TYPE (* A cloud representation for the Arrowhead framework 4.0 *)
  (* Standard: 61499-2 *)
  (* Version 1.0, 2018-09-26, Jose Cabral, fortiss GmbH *)
  (* ASN.1 tag APPLICATION 1 *)
  ArrowheadCloud : STRUCT
    operator : WSTRING;
    cloudName : WSTRING; (* Name of the cloud *)
    address : WSTRING;
    port : DINT;
    gatekeeperServiceURI : WSTRING;
    authenticationInfo : WSTRING;
    secure : BOOL;
  END_STRUCT;
END_TYPE
